# EPICS substitutions: evrSupport/Db/ioc/evrXL16.substitutions
#==============================================================================
#
# Abs:  LCLS EVR IOC records for IOC XL16
#
# Name: evrXL16.substitutions
#
# Note: Signal names must be all uppercase and 12 chars or less to follow
#       LCLS naming conventions.
#
# Macros:
# Set LOCA to 4 char location name.
#
# For VME EVR modules, CARD must be set to the physical slot in the crate
# where the EVR resides, starting from 1.  For PMC EVR modules, CARD must
# be 0 for slot 1 and 1 for slot 2.
#
#==============================================================================
#
file evr.db
{
# PRIM = EVR
# UNIT = xx01 for first EVR in crate, UNIT = xx02 for second EVR, etc.
#     where xx = subsystem ID.
#                               Default Pulse
#	 Location Unit   Card   Delay   Width (clock ticks)
pattern { LOCA  , UNIT , CARD , DELAY , WIDTH }
	{ XL16  , EV01 ,  0   ,   8   ,  13   }
	{ XL16  , EV02 ,  1   ,   8   ,  13   }
	{ XL16  , EV03 ,  2   ,   8   ,  13   }
}
file evrEvent.db
{
# PRIM = EVR
# UNIT = xx01 for first EVR in card, UNIT = xx02 for second EVR, etc.
#
#	 Location Unit   Card  <----------------------------  Event -------------------------->
pattern { LOCA  , UNIT , CARD , NAME    , ID ,P0,P1,P2,P3,P4,P5,P6,P7,P8,P9,P10,P11,P12,P13,VME}
	{ XL16  , EV01 ,   0  , EVENT1  , 1  , 0, 0, 0, 0, 0, 0, 0, 0, 0, 0, 0 , 0 , 0 , 0 , 1 }
	{ XL16  , EV01 ,   0  , EVENT2  , 2  , 0, 0, 0, 0, 0, 0, 0, 0, 0, 0, 0 , 0 , 0 , 0 , 1 }
	{ XL16  , EV01 ,   0  , EVENT3  , 3  , 0, 0, 0, 0, 0, 0, 0, 0, 0, 0, 0 , 0 , 0 , 0 , 1 }
	{ XL16  , EV01 ,   0  , EVENT4  , 4  , 0, 0, 0, 0, 0, 0, 0, 0, 0, 0, 0 , 0 , 0 , 0 , 1 }
	{ XL16  , EV01 ,   0  , EVENT5  , 5  , 0, 0, 0, 0, 0, 0, 0, 0, 0, 0, 0 , 0 , 0 , 0 , 1 }
	{ XL16  , EV01 ,   0  , EVENT6  , 6  , 0, 0, 0, 0, 0, 0, 0, 0, 0, 0, 0 , 0 , 0 , 0 , 1 }
	{ XL16  , EV01 ,   0  , EVENT7  , 7  , 0, 0, 0, 0, 0, 0, 0, 0, 0, 0, 0 , 0 , 0 , 0 , 1 }
	{ XL16  , EV01 ,   0  , EVENT8  , 8  , 1, 0, 0, 0, 0, 0, 0, 0, 0, 0, 0 , 0 , 0 , 0 , 1 }
	{ XL16  , EV01 ,   0  , EVENT9  , 9  , 0, 0, 0, 0, 0, 0, 0, 0, 0, 0, 0 , 0 , 0 , 0 , 1 }
	{ XL16  , EV01 ,   0  , EVENT10 , 10 , 0, 0, 0, 0, 0, 0, 0, 0, 0, 0, 0 , 0 , 0 , 0 , 1 }
	{ XL16  , EV01 ,   0  , EVENT11 , 11 , 0, 0, 0, 0, 0, 0, 0, 0, 0, 0, 0 , 0 , 0 , 0 , 1 }
	{ XL16  , EV01 ,   0  , EVENT12 , 12 , 0, 0, 0, 0, 0, 0, 0, 0, 0, 0, 0 , 0 , 0 , 0 , 1 }
	{ XL16  , EV01 ,   0  , EVENT13 , 13 , 0, 0, 0, 0, 0, 0, 0, 0, 0, 0, 0 , 0 , 0 , 0 , 1 }
	{ XL16  , EV01 ,   0  , EVENT14 , 14 , 0, 0, 0, 0, 0, 0, 0, 0, 0, 0, 0 , 0 , 0 , 0 , 1 }
	{ XL16  , EV01 ,   0  , EVENT15 , 15 , 0, 0, 0, 0, 0, 0, 0, 0, 0, 0, 0 , 0 , 0 , 0 , 1 }

	{ XL16  , EV02 ,   1  , EVENT1  , 1  , 0, 0, 0, 0, 0, 0, 0, 0, 0, 0, 0 , 0 , 0 , 0 , 0 }
	{ XL16  , EV02 ,   1  , EVENT2  , 2  , 0, 0, 0, 0, 0, 0, 0, 0, 0, 0, 0 , 0 , 0 , 0 , 0 }
	{ XL16  , EV02 ,   1  , EVENT3  , 3  , 0, 0, 0, 0, 0, 0, 0, 0, 0, 0, 0 , 0 , 0 , 0 , 0 }
	{ XL16  , EV02 ,   1  , EVENT4  , 4  , 0, 0, 0, 0, 0, 0, 0, 0, 0, 0, 0 , 0 , 0 , 0 , 0 }
	{ XL16  , EV02 ,   1  , EVENT5  , 5  , 0, 0, 0, 0, 0, 0, 0, 0, 0, 0, 0 , 0 , 0 , 0 , 0 }
	{ XL16  , EV02 ,   1  , EVENT6  , 6  , 0, 0, 0, 0, 0, 0, 0, 0, 0, 0, 0 , 0 , 0 , 0 , 0 }
	{ XL16  , EV02 ,   1  , EVENT7  , 7  , 0, 0, 0, 0, 0, 0, 0, 0, 0, 0, 0 , 0 , 0 , 0 , 0 }
	{ XL16  , EV02 ,   1  , EVENT8  , 8  , 1, 0, 0, 0, 0, 0, 0, 0, 0, 0, 0 , 0 , 0 , 0 , 0 }
	{ XL16  , EV02 ,   1  , EVENT9  , 9  , 0, 0, 0, 0, 0, 0, 0, 0, 0, 0, 0 , 0 , 0 , 0 , 0 }
	{ XL16  , EV02 ,   1  , EVENT10 , 10 , 0, 0, 0, 0, 0, 0, 0, 0, 0, 0, 0 , 0 , 0 , 0 , 0 }
	{ XL16  , EV02 ,   1  , EVENT11 , 11 , 0, 0, 0, 0, 0, 0, 0, 0, 0, 0, 0 , 0 , 0 , 0 , 0 }
	{ XL16  , EV02 ,   1  , EVENT12 , 12 , 0, 0, 0, 0, 0, 0, 0, 0, 0, 0, 0 , 0 , 0 , 0 , 0 }
	{ XL16  , EV02 ,   1  , EVENT13 , 13 , 0, 0, 0, 0, 0, 0, 0, 0, 0, 0, 0 , 0 , 0 , 0 , 0 }
	{ XL16  , EV02 ,   1  , EVENT14 , 14 , 0, 0, 0, 0, 0, 0, 0, 0, 0, 0, 0 , 0 , 0 , 0 , 0 }
	{ XL16  , EV02 ,   1  , EVENT15 , 15 , 0, 0, 0, 0, 0, 0, 0, 0, 0, 0, 0 , 0 , 0 , 0 , 0 }

	{ XL16  , EV03 ,   2  , EVENT1  , 1  , 0, 0, 0, 0, 0, 0, 0, 0, 0, 0, 0 , 0 , 0 , 0 , 0 }
	{ XL16  , EV03 ,   2  , EVENT2  , 2  , 0, 0, 0, 0, 0, 0, 0, 0, 0, 0, 0 , 0 , 0 , 0 , 0 }
	{ XL16  , EV03 ,   2  , EVENT3  , 3  , 0, 0, 0, 0, 0, 0, 0, 0, 0, 0, 0 , 0 , 0 , 0 , 0 }
	{ XL16  , EV03 ,   2  , EVENT4  , 4  , 0, 0, 0, 0, 0, 0, 0, 0, 0, 0, 0 , 0 , 0 , 0 , 0 }
	{ XL16  , EV03 ,   2  , EVENT5  , 5  , 0, 0, 0, 0, 0, 0, 0, 0, 0, 0, 0 , 0 , 0 , 0 , 0 }
	{ XL16  , EV03 ,   2  , EVENT6  , 6  , 0, 0, 0, 0, 0, 0, 0, 0, 0, 0, 0 , 0 , 0 , 0 , 0 }
	{ XL16  , EV03 ,   2  , EVENT7  , 7  , 0, 0, 0, 0, 0, 0, 0, 0, 0, 0, 0 , 0 , 0 , 0 , 0 }
	{ XL16  , EV03 ,   2  , EVENT8  , 8  , 1, 0, 0, 0, 0, 0, 0, 0, 0, 0, 0 , 0 , 0 , 0 , 0 }
	{ XL16  , EV03 ,   2  , EVENT9  , 9  , 0, 0, 0, 0, 0, 0, 0, 0, 0, 0, 0 , 0 , 0 , 0 , 0 }
	{ XL16  , EV03 ,   2  , EVENT10 , 10 , 0, 0, 0, 0, 0, 0, 0, 0, 0, 0, 0 , 0 , 0 , 0 , 0 }
	{ XL16  , EV03 ,   2  , EVENT11 , 11 , 0, 0, 0, 0, 0, 0, 0, 0, 0, 0, 0 , 0 , 0 , 0 , 0 }
	{ XL16  , EV03 ,   2  , EVENT12 , 12 , 0, 0, 0, 0, 0, 0, 0, 0, 0, 0, 0 , 0 , 0 , 0 , 0 }
	{ XL16  , EV03 ,   2  , EVENT13 , 13 , 0, 0, 0, 0, 0, 0, 0, 0, 0, 0, 0 , 0 , 0 , 0 , 0 }
	{ XL16  , EV03 ,   2  , EVENT14 , 14 , 0, 0, 0, 0, 0, 0, 0, 0, 0, 0, 0 , 0 , 0 , 0 , 0 }
	{ XL16  , EV03 ,   2  , EVENT15 , 15 , 0, 0, 0, 0, 0, 0, 0, 0, 0, 0, 0 , 0 , 0 , 0 , 0 }
}
file evrEventRate.db
{
# PRIM = IOC
# UNIT = xxyy, where xx = subsystem ID and yy=index of that subsystem in LOCA.
#
#	 Location Unit   Card
pattern { LOCA  , UNIT , CARD , NAME    , ID , FLNK                     }
	{ XL16  , EV01 ,   0  , EVENT1  , 1  , "IOC:XL16:EV01:FIDUCIAL" }
	{ XL16  , EV01 ,   0  , EVENT2  , 2  , ""                       }
	{ XL16  , EV01 ,   0  , EVENT3  , 3  , ""                       }
	{ XL16  , EV01 ,   0  , EVENT4  , 4  , ""                       }
	{ XL16  , EV01 ,   0  , EVENT5  , 5  , ""                       }
	{ XL16  , EV01 ,   0  , EVENT6  , 6  , ""                       }
	{ XL16  , EV01 ,   0  , EVENT7  , 7  , ""                       }
	{ XL16  , EV01 ,   0  , EVENT8  , 8  , ""                       }
	{ XL16  , EV01 ,   0  , EVENT9  , 9  , ""                       }
	{ XL16  , EV01 ,   0  , EVENT10 , 10 , ""                       }
	{ XL16  , EV01 ,   0  , EVENT11 , 11 , ""                       }
	{ XL16  , EV01 ,   0  , EVENT12 , 12 , ""                       }
	{ XL16  , EV01 ,   0  , EVENT13 , 13 , ""                       }
	{ XL16  , EV01 ,   0  , EVENT14 , 14 , ""                       }
	{ XL16  , EV01 ,   0  , EVENT15 , 15 , ""                       }
}
